// TIA Portal project "Motor Control" (V16)

(* hardware
DEVICE "S71500/ET200MP station_1"  S7-1500 station
   slot 0: "Rail_0"  Rack  6ES7 590-1***0-0AA0
   slot 1: "PLC_1"  CPU 1516-3 PN/DP  6ES7 516-3AN00-0AB0  V1.8
      slot 3: "CPU display_1"  6ES7591-1BA00-0AA0
      slot 32768: "PROFINET interface_1"  X1
         slot 32769: "Port_1"  X1 P1
         slot 32770: "Port_2"  X1 P2
      slot 33024: "PROFINET interface_2"  X2
         slot 33025: "Port_1"  X2 P1
      slot 33280: "DP interface_1"  X3
DEVICE "HMI_1"  TP900 Comfort
   slot 0: "HMI_1"  TP900 Comfort  6AV2 124-0JC01-0AX0  16.0.0.0
   slot 1: "HMI_RT_1"  TP900 Comfort  6AV2 124-0JC01-0AX0  16.0.0.0
   slot 5: "HMI_1.IE_CP_1"  PROFINET Interface  16.0.0.0
      slot 1: "PROFINET Interface_1"  PROFINET Interface
         slot 1: "Port_1"  Port
         slot 2: "Port_2"  Port
   slot 7: "HMI_1.MPI/DP_CP_1"  MPI/DP Interface  16.0.0.0
*)

// ===== PLC "PLC_1"  CPU 1516-3 PN/DP =====

VAR_GLOBAL   // PLC tag table "Default tag table"
   "Start" AT %M0.0 : Bool;
   "Motor1" AT %M0.1 : Bool;
   "Motor2" AT %M0.2 : Bool;
   "0 ms" AT %MD2 : Time;
   "Motor3" AT %M0.3 : Bool;
   "Stop" AT %M0.4 : Bool;
   "Deneme" AT %M0.5 : Bool;
   "PTRIG" AT %M0.6 : Bool;
   "PTRIG1" AT %M0.7 : Bool;
   "PTRIG2" AT %M1.0 : Bool;
   "PTRIG3" AT %M1.1 : Bool;
   "PTRIG4" AT %M1.2 : Bool;
   "PTRIG5" AT %M1.3 : Bool;
   "PTRIG6" AT %M1.4 : Bool;
   "STOP_BASILDI" AT %M1.5 : Bool;
   "START_VERILDI" AT %M1.6 : Bool;
END_VAR

DATA_BLOCK "Zamanlayıcı"   // DB1
{ S7_Optimized_Access := 'TRUE' }
VERSION : 0.1
   VAR
      "1.M Start" : Int;
      "2.M Start" : Int;
   END_VAR
BEGIN
END_DATA_BLOCK

// folder: System blocks/Program resources

DATA_BLOCK "IEC_Timer_0_DB_1"   // DB3
{ S7_Optimized_Access := 'TRUE' }
AUTHOR : Simatic
FAMILY : IEC
NAME : IEC_TMR
VERSION : 1.0
// stored: InstanceOfName IEC_TIMER
"IEC_TIMER"
BEGIN
END_DATA_BLOCK

DATA_BLOCK "IEC_Timer_0_DB_2"   // DB4
{ S7_Optimized_Access := 'TRUE' }
AUTHOR : Simatic
FAMILY : IEC
NAME : IEC_TMR
VERSION : 1.0
// stored: InstanceOfName IEC_TIMER
"IEC_TIMER"
BEGIN
END_DATA_BLOCK

DATA_BLOCK "IEC_Timer_0_DB_3"   // DB5
{ S7_Optimized_Access := 'TRUE' }
AUTHOR : Simatic
FAMILY : IEC
NAME : IEC_TMR
VERSION : 1.0
// stored: InstanceOfName IEC_TIMER
"IEC_TIMER"
BEGIN
END_DATA_BLOCK

DATA_BLOCK "IEC_Timer_0_DB_4"   // DB6
{ S7_Optimized_Access := 'TRUE' }
AUTHOR : Simatic
FAMILY : IEC
NAME : IEC_TMR
VERSION : 1.0
// stored: InstanceOfName IEC_TIMER
"IEC_TIMER"
BEGIN
END_DATA_BLOCK

// folder: (top level)

ORGANIZATION_BLOCK "Main"   // OB1, LAD, ProgramCycle
TITLE = "Main Program Sweep (Cycle)"
{ S7_Optimized_Access := 'TRUE' }
VERSION : 0.1
   VAR_INPUT
      Initial_Call : Bool;   // Initial call of this OB
      Remanence : Bool;   // =True, if remanent data are available
   END_VAR
   VAR_TEMP   // added for the SCL form of the ladder/FBD networks
      _w1 : Bool;
      _w2 : Bool;
      _w3 : Bool;
   END_VAR
BEGIN

REGION Network 1
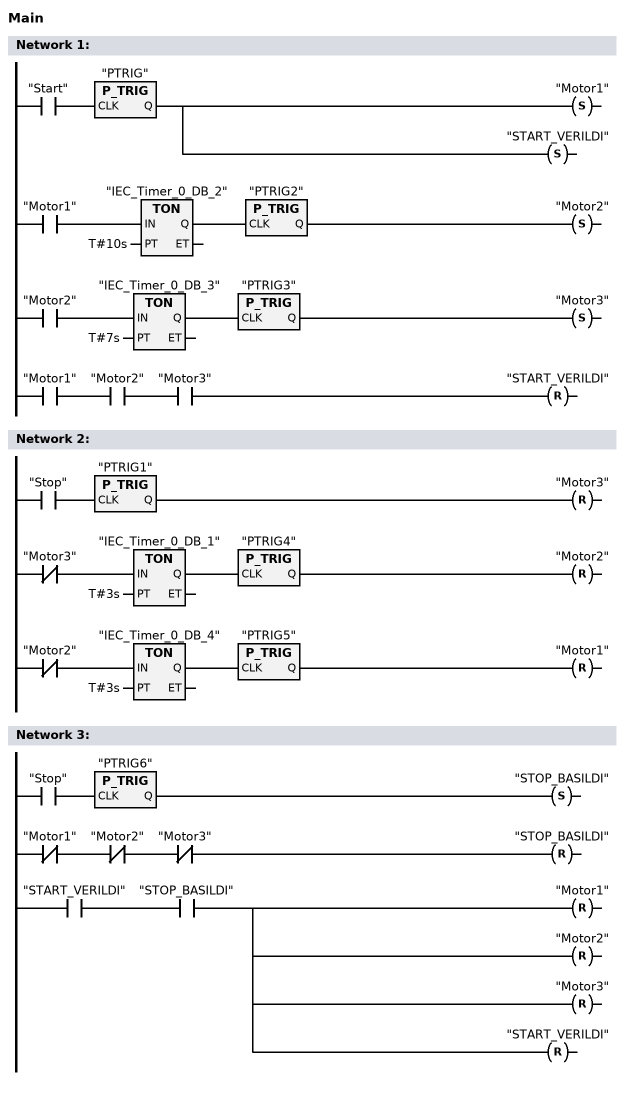
   #_w1 := "Start" AND NOT "PTRIG";   // rising edge
   "PTRIG" := "Start";
   IF #_w1 THEN
       "Motor1" := TRUE;
       "START_VERILDI" := TRUE;
   END_IF;
   "IEC_Timer_0_DB_2".TON(IN := "Motor1", PT := T#10s);
   #_w2 := "IEC_Timer_0_DB_2".Q AND NOT "PTRIG2";   // rising edge
   "PTRIG2" := "IEC_Timer_0_DB_2".Q;
   IF #_w2 THEN "Motor2" := TRUE; END_IF;
   "IEC_Timer_0_DB_3".TON(IN := "Motor2", PT := T#7s);
   #_w3 := "IEC_Timer_0_DB_3".Q AND NOT "PTRIG3";   // rising edge
   "PTRIG3" := "IEC_Timer_0_DB_3".Q;
   IF #_w3 THEN "Motor3" := TRUE; END_IF;
   IF "Motor1" AND "Motor2" AND "Motor3" THEN "START_VERILDI" := FALSE; END_IF;
END_REGION

REGION Network 2
   #_w1 := "Stop" AND NOT "PTRIG1";   // rising edge
   "PTRIG1" := "Stop";
   IF #_w1 THEN "Motor3" := FALSE; END_IF;
   "IEC_Timer_0_DB_1".TON(IN := NOT "Motor3", PT := T#3s);
   #_w2 := "IEC_Timer_0_DB_1".Q AND NOT "PTRIG4";   // rising edge
   "PTRIG4" := "IEC_Timer_0_DB_1".Q;
   IF #_w2 THEN "Motor2" := FALSE; END_IF;
   "IEC_Timer_0_DB_4".TON(IN := NOT "Motor2", PT := T#3s);
   #_w3 := "IEC_Timer_0_DB_4".Q AND NOT "PTRIG5";   // rising edge
   "PTRIG5" := "IEC_Timer_0_DB_4".Q;
   IF #_w3 THEN "Motor1" := FALSE; END_IF;
END_REGION

REGION Network 3
   RUNG wire#powerrail
      Contact( "Stop" )
      P_Trig( "PTRIG6" )
      S_Coil( "STOP_BASILDI" )
   END_RUNG
   RUNG wire#powerrail
      I_Contact( "Motor1" )
      I_Contact( "Motor2" )
      I_Contact( "Motor3" )
      R_Coil( "STOP_BASILDI" )
   END_RUNG
   RUNG wire#powerrail
      Contact( "START_VERILDI" )
      Contact( "STOP_BASILDI" )
      wire#w1
      R_Coil( "Motor1" )
   END_RUNG
   RUNG wire#w1
      R_Coil( "Motor2" )
   END_RUNG
   RUNG wire#w1
      R_Coil( "Motor3" )
   END_RUNG
   RUNG wire#w1
      R_Coil( "START_VERILDI" )
   END_RUNG
   // the same network as SCL:
   #_w1 := "Stop" AND NOT "PTRIG6";   // rising edge
   "PTRIG6" := "Stop";
   IF #_w1 THEN "STOP_BASILDI" := TRUE; END_IF;
   IF NOT "Motor1" AND NOT "Motor2" AND NOT "Motor3" THEN "STOP_BASILDI" := FALSE; END_IF;
   IF "START_VERILDI" AND "STOP_BASILDI" THEN
       "Motor1" := FALSE;
       "Motor2" := FALSE;
       "Motor3" := FALSE;
       "START_VERILDI" := FALSE;
   END_IF;
END_REGION
END_ORGANIZATION_BLOCK

(* ===== HMI "HMI_RT_1" =====
system functions are stored by id; their names below are inferred from use
connection "HMI_Connection_1": ETHERNET, S7_1500_OMS

HMI tags "Default tag table"
   "Tag_ScreenNumber" : UInt, internal
   "Motor1" : Bool = PLC Motor1 AT %M0.1, 1 s
   "Motor2" : Bool = PLC Motor2 AT %M0.2, 1 s
   "Motor3" : Bool = PLC Motor3 AT %M0.3, 1 s
   "Start" : Bool = PLC Start AT %M0.0, 1 s
   "Stop" : Bool = PLC Stop AT %M0.4, 1 s

screen "Root screen" 800x420, template "Template_1"
   on GenerateScreen: SetTag("Tag_ScreenNumber", 1)
   TextField "Text field_1" at 208,83 size 82x28; Text '1.Motor'
   TextField "Text field_2" at 207,132 size 77x28; Text '2.Motor'
   TextField "Text field_3" at 210,195 size 77x28; Text '3.Motor'
   Circle "Circle_1" at 352,75 size 48x48
      Appearance <- "Motor1"
   Circle "Circle_2" at 352,126 size 48x48
      Appearance <- "Motor2"
   Circle "Circle_3" at 352,178 size 48x48
      Appearance <- "Motor3"
   Button "Button_1" at 227,10 size 96x32; TextOff 'START'
      on Press: function_b14e0dd5("Start", 0)
   Button "Button_2" at 376,9 size 96x32; TextOff 'STOP'
      on Press: function_b14e0dd5("Stop", 0)

Template "Template_1" 800x420
   Button "Exit" at 720,360 size 78x58; TextOff 'Exit'; PictureOff "ExitRuntime_TP900_Comfort_TR"; PictureOn "ExitRuntime_TP900_Comfort_TR"
      on Release: StopRuntime(0)
   Button "Template_Button" at 640,360 size 78x58; TextOff 'Text'
   Button "Template_Button_1" at 560,360 size 78x58; TextOff 'Text'
   Button "Template_Button_2" at 480,360 size 78x58; TextOff 'Text'
   Button "Template_Button_3" at 400,360 size 78x58; TextOff 'Text'
   Button "Template_Button_4" at 321,360 size 78x58; TextOff 'Text'
   Button "Template_Button_5" at 241,360 size 78x58; TextOff 'Text'
   Button "Template_Button_6" at 161,360 size 78x58; TextOff 'Text'
   Button "Alarms" at 81,360 size 78x58; TextOff 'Alarms'; PictureOff "AlarmDisplay_TP900_Comfort_TR"; PictureOn "AlarmDisplay_TP900_Comfort_TR"
      on Release: function_ef3f5d25("Alarm window_Unacknowledged", -1)
   Button "Start screen" at 1,360 size 78x58; TextOff 'Start screen'; PictureOff "NavigateHome_TP900_Comfort_TR"; PictureOn "NavigateHome_TP900_Comfort_TR"
      on Release: ActivateScreen("Root screen", 0)
*)